(****************************************************************************************)
(*							Beckhoff Automation Poland									*)
(*								FB_SaveLineToFile  v2.0									*)
(*									26.06.2014											*)
(*						Blok funkcyjny zapisujacy tekst do pliku						*)
(*______________________________________________________________________________________
	Versions:
		v1.1	05.08.2016	* Przepisana wersja do TwinCat3
		v1.0	17.09.2012	* Podstawowa wersja z TwinCat2
________________________________________________________________________________________*)
FUNCTION_BLOCK FB_SaveTextToFile
VAR_INPUT
	bExecute		: BOOL;			(* Komenda wpisu *)
	AmsNetId		: T_AmsNetId;	(* AMS NET ID obiektu docelowego, gdy lokalnie, to zmienna moze byc pusta *)
	sPath			: STRING; 		(* Sciezka pliku, np  'Hard Disk\'*)
	sName			: STRING; 		(* Nazwa pliku wraz z rozszerzeniem 'LogFile.txt'; *)
	sLine			: STRING;		(* Tresc wpisu *)
END_VAR

VAR_OUTPUT
	bBusy		: BOOL;
	bError		: BOOL;
END_VAR
VAR
	fbFileOpen	: FB_FileOpen;
	ftOpen		: F_TRIG;
	fbFilePuts	: FB_FilePuts;
	ftPuts		: F_TRIG;
	fbFileClose	: FB_FileClose;
	ftClose		: F_TRIG;
END_VAR
VAR // added by the converter: edge detectors and wires of the graphical bodies
    _w1 : BOOL;
END_VAR

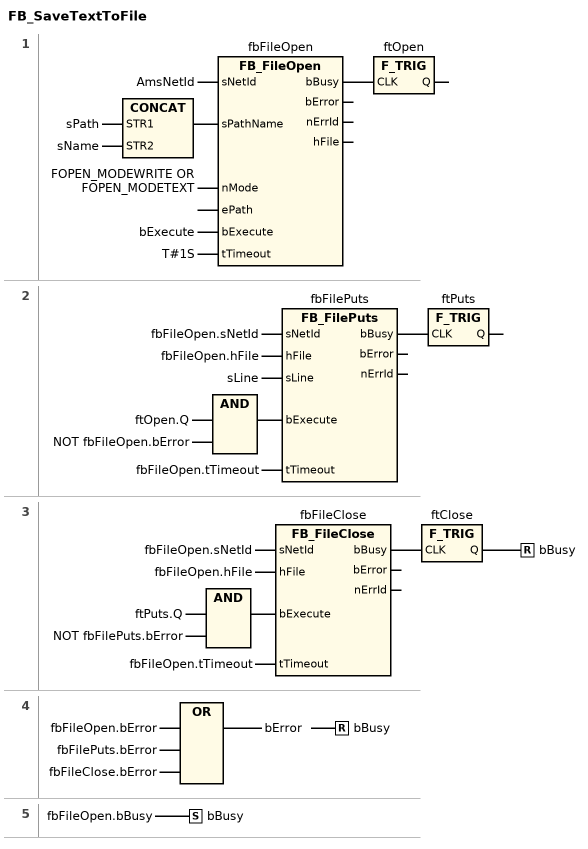
// NETWORK 1
fbFileOpen(
    sNetId := AmsNetId,
    sPathName := CONCAT(STR1 := sPath, STR2 := sName),
    nMode := FOPEN_MODEWRITE OR FOPEN_MODETEXT,
    bExecute := bExecute,
    tTimeout := T#1S); // FB_FileOpen
ftOpen(CLK := fbFileOpen.bBusy); // F_TRIG

// NETWORK 2
fbFilePuts(
    sNetId := fbFileOpen.sNetId,
    hFile := fbFileOpen.hFile,
    sLine := sLine,
    bExecute := ftOpen.Q AND (NOT fbFileOpen.bError),
    tTimeout := fbFileOpen.tTimeout); // FB_FilePuts
ftPuts(CLK := fbFilePuts.bBusy); // F_TRIG

// NETWORK 3
fbFileClose(
    sNetId := fbFileOpen.sNetId,
    hFile := fbFileOpen.hFile,
    bExecute := ftPuts.Q AND (NOT fbFilePuts.bError),
    tTimeout := fbFileOpen.tTimeout); // FB_FileClose
ftClose(CLK := fbFileClose.bBusy); // F_TRIG
bBusy R= ftClose.Q;

// NETWORK 4
_w1 := fbFileOpen.bError OR fbFilePuts.bError OR fbFileClose.bError;
bError := _w1;
bBusy R= _w1;

// NETWORK 5
bBusy S= fbFileOpen.bBusy;

END_FUNCTION_BLOCK

(* stored: Version 1.1.0.1, ProductVersion 3.1.4026.13, FileIdentifier 674578da8829bb4f1a9f52402103bda0f96f0702, FileSignature 0d08f7a08cb438858e3a5e43a0bbca853cad366c310030bc19b9a083e704626a28b4db2466cde4358d47145bdb9d5dc595bedcbbf0ce2c884b92a419fccbfe5b130d9e09a29ec22fc557f3c1034641a122814eef8e9aa5b682fac9146567987ade5ab7eb52393d762447fe91d1fe52d1a3799c24c3cee1c8fdd80099877c95e579ef272bf13a46295a5cac6ca42f35f38348337faf3f85a57492bbe306fc88ed6ce90acb5ac0b225df55f75d8c6c0a9f6346b47ea1650b7bd2395c4547e0b2f8327a7c486331411867a05c8931d84f4498b9d61df8b93af44df1cc33275c783acb0cb1d543b962ebae358a2d651fe5b349d1789a12f2c4395da80d3928b5ebb1
   POU FB_SaveTextToFile: Id {cf11fea1-dcc4-422b-8e53-58a6814e398d}, SpecialFunc None *)
